FUNCTION_BLOCK FB_Motor

VAR
	aInputTargets : ARRAY[1..10] OF INT;	

	ThisMotor : FB_XenaxAxisForceFeedback;
	motorParameters : ST_MOTION_PARAMS;
	
	// Movement states for the motor
	enumStates : (INITIALIZE_VALUES, INITIALIZE, FETCH, MOVING, WAIT, GET_NEXT_TARGET, MOVE_TO_TARGET);
	
END_VAR


mStates(); // keep running through states
// ^^ could have manager to have a stack to follow commands
// but for this purpose, its ok

METHOD mInitialize : BOOL

VAR_INPUT
	aInputArray : ARRAY[1..10] OF INT;
END_VAR
aInputTargets := aInputArray;
END_METHOD

METHOD mStates : BOOL

VAR_INPUT
END_VAR

VAR_INST
	// Track index location of input array & value at current index of input array
	nTargetIndex : INT := 1;
	nTargetValue : INT := 0;
	
	// Wait timer between move commands
	tonWaitTimer : TON := (PT := T#500MS);
END_VAR
Thismotor(usiRefernceDirection := INT_TO_USINT(E_JS_MC_REF_MODE.Positive));

CASE enumStates OF
	INITIALIZE_VALUES:
		motorParameters.TargetPos := 0;
		motorParameters.Jerk := 20000;
		motorParameters.TargetAccel := 2000;
		motorParameters.TargetDecel := 2000;
		motorParameters.TargetVel := 1000;
		enumStates := INITIALIZE;
		
		
	INITIALIZE:
		ThisMotor.Initialize(TRUE);
		IF ThisMotor.DidInitialize THEN
			nTargetValue := 0;
			enumStates := MOVE_TO_TARGET;
		END_IF
		
		
	MOVING:
		ThisMotor.MoveAbs(Execute := TRUE, MotionParams := motorParameters);
		IF ThisMotor.DidMoveAbs THEN
			ThisMotor.MoveAbs(Execute := FALSE, MotionParams := motorParameters);
			enumStates := WAIT;
		END_IF
		
		
	WAIT:
		tonWaitTimer(IN := TRUE);
		
		IF tonWaitTimer.Q THEN
			tonWaitTimer(IN := FALSE);
			enumStates := GET_NEXT_TARGET;
		END_IF

		
	GET_NEXT_TARGET:
		
		IF nTargetIndex + 1 > UINT_TO_INT(SIZEOF(aInputTargets)/2) THEN // divide by 2 since the array type is of int (2 bytes per entry)
			nTargetIndex := 1;
		END_IF

		nTargetValue := aInputTargets[nTargetIndex];
		
		nTargetIndex := nTargetIndex + 1;
		
		enumStates := MOVE_TO_TARGET;
		
		
	MOVE_TO_TARGET:
		motorParameters.TargetPos := nTargetValue;
		enumStates := MOVING;
		
END_CASE
END_METHOD

END_FUNCTION_BLOCK

(* stored: Version 1.1.0.1, ProductVersion 3.1.4024.12
   POU FB_Motor: Id {c547f712-1e26-4765-80bd-73a5ca39fd11}, SpecialFunc None
   Method mInitialize: Id {d0d87515-1fa6-436d-af8c-2f33466bfee2}
   Method mStates: Id {1dc201df-a37e-41a0-883b-52165c62b3e7} *)
